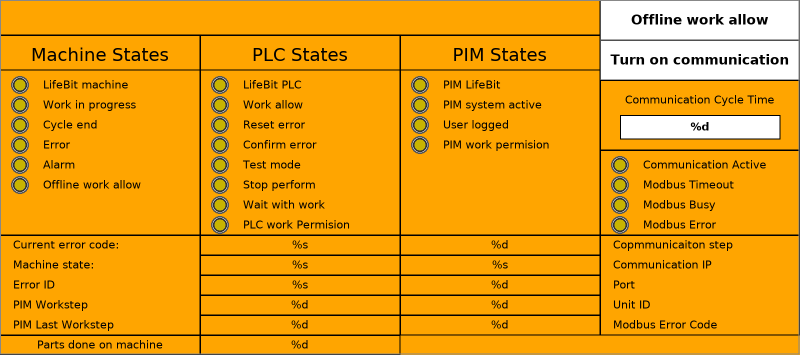
VISUALIZATION vChiniseMachineStatus  // 800x355
VAR_IN_OUT
	stData					:	stPimMachineData;
	fbPIM 					:	fbPIM_Station_V3;
	iActualMachine			: 	UINT;
	fbModbusTCP				:	fbDataExchangePIM;
	bTurnOnCommunication	: 	BOOL;
	iCommunicationCycleTime	: INT;
END_VAR
    Rectangle (600,150 200x85)
    Rectangle (0,235 200x100)
    Rectangle (0,35 200x200)
    Rectangle (0,35 600x35)
    Rectangle (400,35 200x200)
    Rectangle (200,35 200x200)
    Lamp1 (10,75 20x20), variable: stData.bLifeBitMachine, style: Lamp-Lamp1-Yellow
    Label (40,75 150x20), "LifeBit machine"
    Label (5,40 190x30), "Machine States"
    Lamp1 (10,95 20x20), variable: stData.bWorkInProgress, style: Lamp-Lamp1-Yellow
    Label (40,95 150x20), "Work in progress"
    Lamp1 (10,115 20x20), variable: stData.bCycleEnd, style: Lamp-Lamp1-Yellow
    Label (40,115 150x20), "Cycle end"
    Lamp1 (10,135 20x20), variable: stData.bError, style: Lamp-Lamp1-Yellow
    Label (40,135 150x20), "Error"
    Lamp1 (10,155 20x20), variable: stData.bAlarm, style: Lamp-Lamp1-Yellow
    Label (40,155 150x20), "Alarm"
    Lamp1 (10,175 20x20), variable: stData.bOfflineWorkAllow, style: Lamp-Lamp1-Yellow
    Label (40,175 150x20), "Offline work allow"
    Lamp1 (210,75 20x20), variable: stData.bLifeBitPLC, style: Lamp-Lamp1-Yellow
    Label (240,75 150x20), "LifeBit PLC"
    Label (205,40 190x30), "PLC States"
    Lamp1 (210,95 20x20), variable: stData.bWorkAllow, style: Lamp-Lamp1-Yellow
    Label (240,95 150x20), "Work allow"
    Lamp1 (210,115 20x20), variable: stData.bResetError, style: Lamp-Lamp1-Yellow
    Label (240,115 150x20), "Reset error"
    Lamp1 (210,135 20x20), variable: stData.bConfirmError, style: Lamp-Lamp1-Yellow
    Label (240,135 150x20), "Confirm error"
    Lamp1 (210,155 20x20), variable: stData.bTestMode, style: Lamp-Lamp1-Yellow
    Label (240,155 150x20), "Test mode"
    Lamp1 (210,175 20x20), variable: stData.bStopPerform, style: Lamp-Lamp1-Yellow
    Label (240,175 150x20), "Stop perform"
    Lamp1 (210,195 20x20), variable: stData.bWaitWithWork, style: Lamp-Lamp1-Yellow
    Label (240,195 150x20), "Wait with work"
    Lamp1 (410,75 20x20), variable: fbPIM.bPIM_Working, style: Lamp-Lamp1-Yellow
    Label (440,75 150x20), "PIM LifeBit"
    Label (405,40 190x30), "PIM States"
    Lamp1 (410,95 20x20), variable: fbPIM.stPimInOut.bPIMActive, style: Lamp-Lamp1-Yellow
    Label (440,95 150x20), "PIM system active"
    Lamp1 (410,115 20x20), variable: fbPIM.stPimInOut.bUserLogged, style: Lamp-Lamp1-Yellow
    Label (440,115 150x20), "User logged"
    Lamp1 (410,135 20x20), variable: NOT fbPIM.stPimInOut.bWorkBlock_PIM, style: Lamp-Lamp1-Yellow
    Label (440,135 150x20), "PIM work permision"
    Rectangle (200,235 200x20), "%s", text variable: fbPIM.stPimInOut.sErrorCodePLC
    Rectangle (200,255 200x20), "%s", text variable: TO_STRING(fbPIM.nMachineState)
    Rectangle (200,275 200x20), "%s", text variable: fbPIM.nErrorID
    Rectangle (200,295 200x20), "%d", text variable: fbPIM.iWorkStep
    Rectangle (200,315 200x20), "%d", text variable: fbPIM.aiPimWorkStepHistoric
    Lamp1 (210,215 20x20), variable: NOT fbPIM.stPimInOut.bWorkBlock_PLC, style: Lamp-Lamp1-Yellow
    Label (240,215 150x20), "PLC work Permision"
    Label (10,235 150x20), "Current error code:"
    Label (10,255 150x20), "Machine state:"
    Label (10,275 150x20), "Error ID"
    Label (10,295 150x20), "PIM Workstep"
    Label (10,315 150x20), "PIM Last Workstep"
    Rectangle (0,0 600x35), text list: 'tlActualMachineName', text index: iActualMachine
    Rectangle (600,0 200x40), "Offline work allow"
        OnMouseClick: toggle stData.bOfflineWorkAllow
    Rectangle (400,235 200x20), "%d", text variable: fbModbusTCP.iCommunicationStep
    Rectangle (400,255 200x20), "%s", text variable: fbModbusTCP.fbModbusTCP.sIPAddr
    Rectangle (400,275 200x20), "%d", text variable: fbModbusTCP.fbModbusTCP.nTCPPort
    Rectangle (400,295 200x20), "%d", text variable: fbModbusTCP.fbModbusTCP.nUnitID
    Rectangle (400,315 200x20), "%d", text variable: fbModbusTCP.fbModbusTCP.nErrId
    Rectangle (600,235 200x100)
    Label (610,235 150x20), "Copmmunicaiton step"
    Label (610,255 150x20), "Communication IP"
    Label (640,195 150x20), "Modbus Busy"
    Label (640,215 150x20), "Modbus Error"
    Label (610,315 150x20), "Modbus Error Code"
    Rectangle (600,40 200x40), "Turn on communication"
        OnMouseClick: toggle bTurnOnCommunication
    Lamp1 (610,215 20x20), variable: fbModbusTCP.fbModbusTCP.bError, style: Lamp-Lamp1-Yellow
    Lamp1 (610,195 20x20), variable: fbModbusTCP.fbModbusTCP.bError, style: Lamp-Lamp1-Yellow
    Label (640,175 150x20), "Modbus Timeout"
    Lamp1 (610,175 20x20), variable: fbModbusTCP.bCommunicationBlockCycleExtended, style: Lamp-Lamp1-Yellow
    Label (610,295 150x20), "Unit ID"
    Label (610,275 150x20), "Port"
    Label (640,155 150x20), "Communication Active"
    Lamp1 (610,155 20x20), variable: fbModbusTCP.bEnableCommunication, style: Lamp-Lamp1-Yellow
    Rectangle (600,80 200x70)
    Rectangle (620,115 160x24), "%d", text variable: iCommunicationCycleTime
        OnMouseClick: write the text variable via Default, format %d
    Label (610,90 180x20), "Communication Cycle Time"
    Rectangle (200,335 200x20), "%d", text variable: stData.wGoodPartsAmount
    Rectangle (0,335 200x20), "Parts done on machine", text variable: fbPIM.aiPimWorkStepHistoric
END_VISUALIZATION

(* stored: Version 1.1.0.1, ProductVersion 3.1.4024.13
   Visu vChiniseMachineStatus: Id {d951909f-24f0-4534-9b16-f0db920f3b11} *)
